// Block: IPC_Send_Buffer_Log_MES

DATA_BLOCK IPC_Send_Buffer_Log_MES
VERSION : 0.1
   NON_RETAIN
   VAR
      lastId : DInt;
      msg : Array[1..LOG_MSG_ITEMS] of IPC_Msg_Generico;
   END_VAR

BEGIN
   // No initialization required
END_DATA_BLOCK
